Omron CX-Programmer project NewProject (CX-Programmer 9.61)

# PLC NewPLC1: CP1E E20

## Global symbols (name address type ; comment)
0.00 BOOL  ; UP
0.01 BOOL  ; DOWN
0.02 BOOL  ; RESET
10.00 BOOL  ; LAMPU1
10.01 BOOL  ; L2
10.02 BOOL  ; L3

## Program NewProgram1 (cyclic task 0)
Local symbols
U CHANNEL

### Section Section1

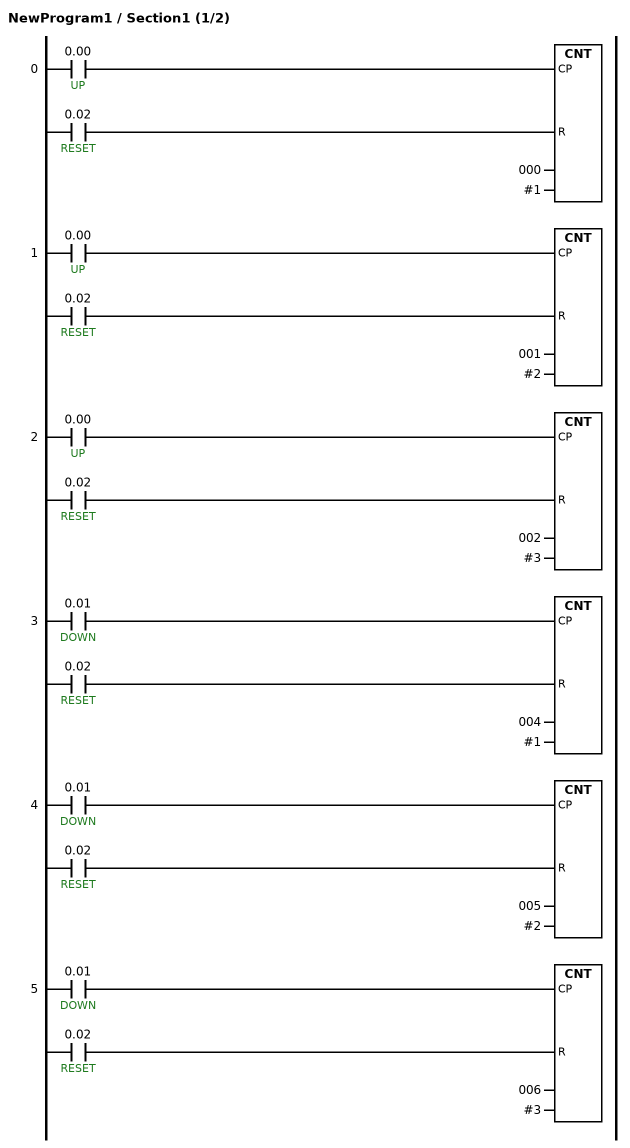
; rung 0
LD 0.00  ; UP
LD 0.02  ; RESET
CNT 000 #1
; rung 1
LD 0.00  ; UP
LD 0.02  ; RESET
CNT 001 #2
; rung 2
LD 0.00  ; UP
LD 0.02  ; RESET
CNT 002 #3
; rung 3
LD 0.01  ; DOWN
LD 0.02  ; RESET
CNT 004 #1
; rung 4
LD 0.01  ; DOWN
LD 0.02  ; RESET
CNT 005 #2
; rung 5
LD 0.01  ; DOWN
LD 0.02  ; RESET
CNT 006 #3

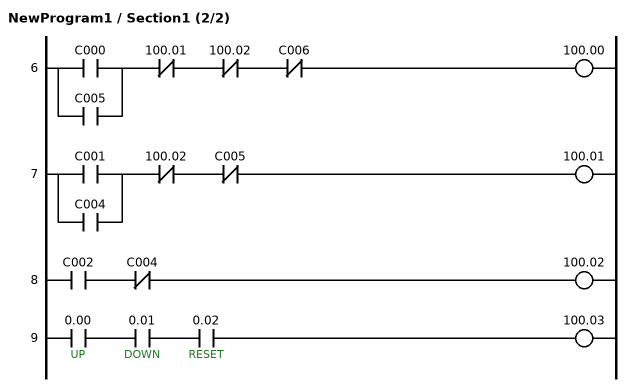
; rung 6
LD C000
OR C005
ANDNOT 100.01
ANDNOT 100.02
ANDNOT C006
OUT 100.00
; rung 7
LD C001
OR C004
ANDNOT 100.02
ANDNOT C005
OUT 100.01
; rung 8
LD C002
ANDNOT C004
OUT 100.02
; rung 9
LD 0.00  ; UP
AND 0.01  ; DOWN
AND 0.02  ; RESET
OUT 100.03

### Section END
; rung 0
END(001)